TYPE Udt_ModuleId :
STRUCT
	nNumber		: UDINT ; // Module identification number used for sorting order
	sName		: STRING; // Module name
	pFunction	: POINTER TO Fb_ModuleBase ;
END_STRUCT
END_TYPE

(* stored: Version 1.1.0.1, ProductVersion 3.1.4024.4
   DUT Udt_ModuleId: Id {478ef210-3e60-456a-8f1e-af63de69c0dd} *)
